(* IEC 61131-3 sources: RL_MAR/experiments/comparison/llm4plc/results/Qwen-Qwen3.5-9B_20260506_150728/20260506_175606, 3 files *)

(* ---- generated_code_iteration_0.st ---- *)
START_ST
FUNCTION_BLOCK FruitJuicingBottling
VAR_INPUT
    StartButton : BOOL; (* Input for starting the process *)
    StopButton : BOOL; (* Input for stopping the process *)
    FruitSelected : BOOL; (* Input indicating fruit selection *)
END_VAR
VAR_OUTPUT
    JuiceProcessing : BOOL; (* Output for controlling juice extraction *)
    BottleFilling : BOOL; (* Output for controlling bottle filling *)
    CapPlacement : BOOL; (* Output for placing caps on bottles *)
    Packaging : BOOL; (* Output for packaging filled bottles *)
    ProcessInProgress : BOOL; (* Indicator for an ongoing process *)
END_VAR
VAR
    state : INT; (* Current FSM State: 0=IDLE, 1=RUNNING, 2=STOPPED *)
    prevState : INT; (* Previous State for transition logic *)
    processInProgress : BOOL; (* Internal variable to track running state *)
END_VAR

(* Initialize state on first execution or reset if needed *)
IF state = 0 AND prevState = 0 THEN
    state := 0;
END_IF;

(* Store current state for next cycle transition logic *)
prevState := state;

(* --- STATE MACHINE LOGIC --- *)

(* Transition from STATE 0 (IDLE) to STATE 1 (RUNNING) *)
(* Condition: StartButton AND FruitSelected AND NOT ProcessInProgress *)
IF state = 0 THEN
    IF StartButton = TRUE AND FruitSelected = TRUE AND ProcessInProgress = FALSE THEN
        state := 1; (* Transition to RUNNING *)
    END_IF;
END_IF;

(* Transition from STATE 1 (RUNNING) to STATE 2 (STOPPED) *)
(* Condition: StopButton OR NOT FruitSelected *)
IF state = 1 THEN
    IF StopButton = TRUE OR FruitSelected = FALSE THEN
        state := 2; (* Transition to STOPPED *)
    END_IF;
END_IF;

(* Transition from STATE 2 (STOPPED) to STATE 0 (IDLE) *)
(* Condition: StopButton is FALSE AND FruitSelected is TRUE *)
IF state = 2 THEN
    IF StopButton = FALSE AND FruitSelected = TRUE THEN
        state := 0; (* Transition back to IDLE *)
    END_IF;
END_IF;

(* --- OUTPUT ASSIGNMENT BASED ON STATE --- *)

(* STATE 0: IDLE *)
IF state = 0 THEN
    JuiceProcessing := FALSE;
    BottleFilling := FALSE;
    CapPlacement := FALSE;
    Packaging := FALSE;
    ProcessInProgress := FALSE;
END_IF;

(* STATE 1: RUNNING *)
IF state = 1 THEN
    JuiceProcessing := TRUE;
    BottleFilling := TRUE;
    CapPlacement := TRUE;
    Packaging := TRUE;
    ProcessInProgress := TRUE;
END_IF;

(* STATE 2: STOPPED *)
IF state = 2 THEN
    JuiceProcessing := FALSE;
    BottleFilling := FALSE;
    CapPlacement := FALSE;
    Packaging := FALSE;
    ProcessInProgress := FALSE;
END_IF;

END_FUNCTION_BLOCK
END_ST

(* ---- generated_code_iteration_1.st ---- *)
START_REASON
The validation feedback indicates a variable naming conflict in the CODESYS compiler. The error message "局部变量 'processInProgress' 已经在'FruitJuicingBottling'中定义" translates to "Local variable 'processInProgress' is already defined in 'FruitJuicingBottling'".

Looking at the provided code:
1. In the `VAR_OUTPUT` section, there is a variable named `ProcessInProgress`.
2. In the `VAR` section, there is a local variable also named `processInProgress` (with different casing).

In IEC 61131-3 Structured Text, variable names are case-insensitive. Therefore, `ProcessInProgress` and `processInProgress` refer to the same identifier. Since `ProcessInProgress` is declared as an output variable, the local variable declaration in the `VAR` section causes a redefinition error.

To fix this, I must remove the duplicate local variable declaration from the `VAR` section. The logic inside the code that references `ProcessInProgress` should continue to use the output variable name (or be consistent), but the declaration causing the conflict must be removed. I will also ensure the logic uses the output variable `ProcessInProgress` directly where appropriate to avoid confusion, though the primary fix is removing the duplicate declaration.
END_REASON

START_ST
FUNCTION_BLOCK FruitJuicingBottling
VAR_INPUT
    StartButton : BOOL; (* Input for starting the process *)
    StopButton : BOOL; (* Input for stopping the process *)
    FruitSelected : BOOL; (* Input indicating fruit selection *)
END_VAR
VAR_OUTPUT
    JuiceProcessing : BOOL; (* Output for controlling juice extraction *)
    BottleFilling : BOOL; (* Output for controlling bottle filling *)
    CapPlacement : BOOL; (* Output for placing caps on bottles *)
    Packaging : BOOL; (* Output for packaging filled bottles *)
    ProcessInProgress : BOOL; (* Indicator for an ongoing process *)
END_VAR
VAR
    state : INT; (* Current FSM State: 0=IDLE, 1=RUNNING, 2=STOPPED *)
    prevState : INT; (* Previous State for transition logic *)
END_VAR

(* Initialize state on first execution or reset if needed *)
IF state = 0 AND prevState = 0 THEN
    state := 0;
END_IF;

(* Store current state for next cycle transition logic *)
prevState := state;

(* --- STATE MACHINE LOGIC --- *)

(* Transition from STATE 0 (IDLE) to STATE 1 (RUNNING) *)
(* Condition: StartButton AND FruitSelected AND NOT ProcessInProgress *)
IF state = 0 THEN
    IF StartButton = TRUE AND FruitSelected = TRUE AND ProcessInProgress = FALSE THEN
        state := 1; (* Transition to RUNNING *)
    END_IF;
END_IF;

(* Transition from STATE 1 (RUNNING) to STATE 2 (STOPPED) *)
(* Condition: StopButton OR NOT FruitSelected *)
IF state = 1 THEN
    IF StopButton = TRUE OR FruitSelected = FALSE THEN
        state := 2; (* Transition to STOPPED *)
    END_IF;
END_IF;

(* Transition from STATE 2 (STOPPED) to STATE 0 (IDLE) *)
(* Condition: StopButton is FALSE AND FruitSelected is TRUE *)
IF state = 2 THEN
    IF StopButton = FALSE AND FruitSelected = TRUE THEN
        state := 0; (* Transition back to IDLE *)
    END_IF;
END_IF;

(* --- OUTPUT ASSIGNMENT BASED ON STATE --- *)

(* STATE 0: IDLE *)
IF state = 0 THEN
    JuiceProcessing := FALSE;
    BottleFilling := FALSE;
    CapPlacement := FALSE;
    Packaging := FALSE;
    ProcessInProgress := FALSE;
END_IF;

(* STATE 1: RUNNING *)
IF state = 1 THEN
    JuiceProcessing := TRUE;
    BottleFilling := TRUE;
    CapPlacement := TRUE;
    Packaging := TRUE;
    ProcessInProgress := TRUE;
END_IF;

(* STATE 2: STOPPED *)
IF state = 2 THEN
    JuiceProcessing := FALSE;
    BottleFilling := FALSE;
    CapPlacement := FALSE;
    Packaging := FALSE;
    ProcessInProgress := FALSE;
END_IF;

END_FUNCTION_BLOCK
END_ST

(* ---- generated_code_iteration_2.st ---- *)
START_REASON
The previous code failed validation due to an encoding issue (GBK codec error at byte 0x80). This typically happens when non-ASCII characters (like Chinese comments or special symbols) are present in the source code but the compiler environment expects ASCII or UTF-8. Additionally, the variable naming conflict identified in the reasoning phase (`ProcessInProgress` in VAR_OUTPUT vs `processInProgress` in VAR) was resolved by removing the duplicate local variable, but the encoding issue is the primary blocker now.

To fix this:
1.  Remove all Chinese comments and replace them with English comments to ensure ASCII compatibility.
2.  Ensure all variable names and logic are strictly ASCII.
3.  Maintain the FUNCTION_BLOCK structure and correct variable scoping (no duplicate `processInProgress` in VAR).
4.  Verify the logic flow for the Finite State Machine (FSM) remains intact.
END_REASON

START_ST
FUNCTION_BLOCK FruitJuicingBottling
VAR_INPUT
    StartButton : BOOL; (* Input for starting the process *)
    StopButton : BOOL; (* Input for stopping the process *)
    FruitSelected : BOOL; (* Input indicating fruit selection *)
END_VAR
VAR_OUTPUT
    JuiceProcessing : BOOL; (* Output for controlling juice extraction *)
    BottleFilling : BOOL; (* Output for controlling bottle filling *)
    CapPlacement : BOOL; (* Output for placing caps on bottles *)
    Packaging : BOOL; (* Output for packaging filled bottles *)
    ProcessInProgress : BOOL; (* Indicator for an ongoing process *)
END_VAR
VAR
    state : INT; (* Current FSM State: 0=IDLE, 1=RUNNING, 2=STOPPED *)
    prevState : INT; (* Previous State for transition logic *)
END_VAR

(* Initialize state on first execution or reset if needed *)
IF state = 0 AND prevState = 0 THEN
    state := 0;
END_IF;

(* Store current state for next cycle transition logic *)
prevState := state;

(* --- STATE MACHINE LOGIC --- *)

(* Transition from STATE 0 (IDLE) to STATE 1 (RUNNING) *)
(* Condition: StartButton AND FruitSelected AND NOT ProcessInProgress *)
IF state = 0 THEN
    IF StartButton = TRUE AND FruitSelected = TRUE AND ProcessInProgress = FALSE THEN
        state := 1; (* Transition to RUNNING *)
    END_IF;
END_IF;

(* Transition from STATE 1 (RUNNING) to STATE 2 (STOPPED) *)
(* Condition: StopButton OR NOT FruitSelected *)
IF state = 1 THEN
    IF StopButton = TRUE OR FruitSelected = FALSE THEN
        state := 2; (* Transition to STOPPED *)
    END_IF;
END_IF;

(* Transition from STATE 2 (STOPPED) to STATE 0 (IDLE) *)
(* Condition: StopButton is FALSE AND FruitSelected is TRUE *)
IF state = 2 THEN
    IF StopButton = FALSE AND FruitSelected = TRUE THEN
        state := 0; (* Transition back to IDLE *)
    END_IF;
END_IF;

(* --- OUTPUT ASSIGNMENT BASED ON STATE --- *)

(* STATE 0: IDLE *)
IF state = 0 THEN
    JuiceProcessing := FALSE;
    BottleFilling := FALSE;
    CapPlacement := FALSE;
    Packaging := FALSE;
    ProcessInProgress := FALSE;
END_IF;

(* STATE 1: RUNNING *)
IF state = 1 THEN
    JuiceProcessing := TRUE;
    BottleFilling := TRUE;
    CapPlacement := TRUE;
    Packaging := TRUE;
    ProcessInProgress := TRUE;
END_IF;

(* STATE 2: STOPPED *)
IF state = 2 THEN
    JuiceProcessing := FALSE;
    BottleFilling := FALSE;
    CapPlacement := FALSE;
    Packaging := FALSE;
    ProcessInProgress := FALSE;
END_IF;

END_FUNCTION_BLOCK
END_ST
